FUNCTION_BLOCK FunkButtons (* Service Interface Function Block Type *)
  (* Standard: SAE J1939; Function: up to 16 Buttons plus START and STOP; Type: LCC 4-6-12-16 Key Remote Control; Description: Copyright (c) 2018, 2023 Jose Cabral, HR Agrartechnik GmbH This program and the accompanying materials are made available under the terms of the Eclipse Public License 2.0 which is available at https://www.eclipse.org/legal/epl-2.0/ SPDX-License-Identifier: EPL-2.0 this maps to IX *)
  (* Version 1.0, 2018-12-05, Jose Cabral *)
  (* Version 1.1, 2022-08-04, Franz Höpfinger, HR Agrartechnik GmbH *)
  (* Version 1.2, 2023-01-05, Franz Höpfinger, HR Agrartechnik GmbH *)
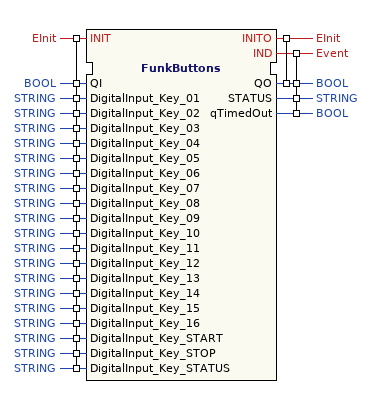
  EVENT_INPUT
    INIT : EInit WITH QI, DigitalInput_Key_01, DigitalInput_Key_02, DigitalInput_Key_03, DigitalInput_Key_04, DigitalInput_Key_05, DigitalInput_Key_06, DigitalInput_Key_07, DigitalInput_Key_08, DigitalInput_Key_09, DigitalInput_Key_10, DigitalInput_Key_11, DigitalInput_Key_12, DigitalInput_Key_13, DigitalInput_Key_14, DigitalInput_Key_15, DigitalInput_Key_16, DigitalInput_Key_START, DigitalInput_Key_STOP, DigitalInput_Key_STATUS; (* Service Initialization *)
  END_EVENT
  EVENT_OUTPUT
    INITO : EInit WITH QO; (* Initialization Confirm *)
    IND WITH QO, STATUS, qTimedOut; (* Indication from Resource *)
  END_EVENT
  VAR_INPUT
    QI : BOOL; (* Event Input Qualifier *)
    DigitalInput_Key_01 : STRING;
    DigitalInput_Key_02 : STRING;
    DigitalInput_Key_03 : STRING;
    DigitalInput_Key_04 : STRING;
    DigitalInput_Key_05 : STRING;
    DigitalInput_Key_06 : STRING;
    DigitalInput_Key_07 : STRING;
    DigitalInput_Key_08 : STRING;
    DigitalInput_Key_09 : STRING;
    DigitalInput_Key_10 : STRING;
    DigitalInput_Key_11 : STRING;
    DigitalInput_Key_12 : STRING;
    DigitalInput_Key_13 : STRING;
    DigitalInput_Key_14 : STRING;
    DigitalInput_Key_15 : STRING;
    DigitalInput_Key_16 : STRING;
    DigitalInput_Key_START : STRING;
    DigitalInput_Key_STOP : STRING;
    DigitalInput_Key_STATUS : STRING;
  END_VAR
  VAR_OUTPUT
    QO : BOOL; (* Event Output Qualifier *)
    STATUS : STRING; (* Service Status *)
    qTimedOut : BOOL;
  END_VAR
END_FUNCTION_BLOCK
